FUNCTION_BLOCK fb_sourcedata (* Event-driven bistable *)
  (* Standard: 61499-1 Annex A; Description: Copyright (c) 2017 fortiss GmbH This program and the accompanying materials are made available under the terms of the Eclipse Public License 2.0 which is available at https://www.eclipse.org/legal/epl-2.0/ SPDX-License-Identifier: EPL-2.0 *)
  (* Version 1.0, 2017-09-22, Alois Zoitl, fortiss GmbH, initial API and implementation and/or initial documentation *)
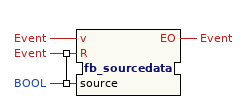
  EVENT_INPUT
    v; (* Set output Q *)
    R WITH source; (* Reset output Q *)
  END_EVENT
  EVENT_OUTPUT
    EO; (* Output Q has changed *)
  END_EVENT
  VAR_INPUT
    source : BOOL;
  END_VAR
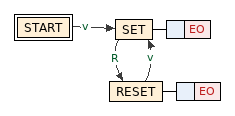
  EC_STATES
    START; (* Initial State *)
    SET : -> EO;
    RESET : -> EO;
  END_STATES
  EC_TRANSITIONS
    START TO SET := v;
    SET TO RESET := R;
    RESET TO SET := v;
  END_TRANSITIONS
END_FUNCTION_BLOCK
